{attribute 'qualified_only'}
VAR_GLOBAL
	// Dewar Temperature sensor error
	Dewar_temperature_error	AT%I*: BOOL;

END_VAR

(* stored: Version 1.1.0.1, ProductVersion 3.1.4024.9
   GVL GVL_Auxiliary: Id {6c7fe825-7173-4b37-8d55-28187f2f4394} *)
